// TIA Portal project "Lab1" (V15)

(* hardware
DEVICE "S7-1200 station_1"  S7-1200 Station
   slot 0: "Rack_0"  S7-1200 Rack  Rack  V1.0
   slot 1: "PLC_1"  CPU 1214C AC/DC/Rly  6ES7 214-1BG40-0XB0  V4.2
DEVICE "HMI_1"  KTP1000 Basic color PN
   slot 0: "HMI_1"  KTP1000 Basic color PN  6AV6 647-0AF11-3AX0  12.0.0.0
   slot 1: "HMI_RT_1"  KTP1000 Basic color PN  6AV6 647-0AF11-3AX0  12.0.0.0
   slot 5: "HMI_1.IE_CP_1"  PROFINET Interface  12.0.0.0
      slot 1: "PROFINET Interface_1"  PROFINET Interface
         slot 1: "Port_1"  Port
*)

// ===== PLC "PLC_1"  CPU 1214C AC/DC/Rly =====

VAR_GLOBAL   // PLC tag table "Default tag table"
   "Start_NC" AT %M4.0 : Bool;
   "Manual_NO" AT %I0.2 : Bool;
   "Auto_NO" AT %I0.3 : Bool;
   "Stop_NC" AT %M4.1 : Bool;
   "SigSklop_NC" AT %I0.6 : Bool;
   "Bimetal_NC" AT %I0.7 : Bool;
   "Prekostruj_NO" AT %I1.0 : Bool;
   "Kontaktor_NO" AT %I1.1 : Bool;
   "Zelena" AT %Q0.0 : Bool;
   "Crvena" AT %Q0.1 : Bool;
   "Kontaktor" AT %Q0.2 : Bool;
   "Clock_Byte" AT %MB53 : Byte;
   "Clock_10Hz" AT %M53.0 : Bool;
   "Clock_5Hz" AT %M53.1 : Bool;
   "Clock_2.5Hz" AT %M53.2 : Bool;
   "Clock_2Hz" AT %M53.3 : Bool;
   "Clock_1.25Hz" AT %M53.4 : Bool;
   "Clock_1Hz" AT %M53.5 : Bool;
   "Clock_0.625Hz" AT %M53.6 : Bool;
   "Clock_0.5Hz" AT %M53.7 : Bool;
   "Blink" AT %M3.2 : Bool;
   "Blink_FF" AT %M3.1 : Bool;
   "Blink_Pulse" AT %M3.0 : Bool;
   "Auto_Stanje_FF" AT %M2.0 : Bool;
   "Greska" AT %M0.4 : Bool;
   "Greska_Bimetal" AT %M0.0 : Bool;
   "Greska_Prekostruj" AT %M0.1 : Bool;
   "Greska_Kontaktor" AT %M0.2 : Bool;
   "Greska_Svestop" AT %M0.3 : Bool;
   "Cekamo" AT %M2.2 : Bool;
   "Blink_Cnt_Greska_Pos" AT %M3.3 : Bool;
   "Blink_FF_Greska_Pos" AT %M3.4 : Bool;
   "OFF_NO" AT %M2.1 : Bool;
   "Bimetal_FF" AT %M1.0 : Bool;
   "Prekostruj_FF" AT %M1.1 : Bool;
   "Svestop_FF" AT %M1.3 : Bool;
   "GKontaktor_FF" AT %M1.2 : Bool;
   "Cekamo_Trig_P" AT %M2.3 : Bool;
   "Cekamo_Trig_N" AT %M2.4 : Bool;
   "Ocekivani_Kontaktor" AT %M2.5 : Bool;
   "Start_Taster_NC" AT %I0.0 : Bool;
   "Stop_Taster_NC" AT %I0.4 : Bool;
   "Start_HMI_NO" AT %M4.2 : Bool;
   "Stop_HMI_NO" AT %M4.3 : Bool;
   "ManualYES" AT %M4.4 : Bool;
   "AlarmWord" AT %MW0 : Word;
END_VAR

// folder: System blocks/Program resources

DATA_BLOCK "Counter_Blink"   // DB1
{ S7_Optimized_Access := 'TRUE' }
AUTHOR : Simatic
FAMILY : IEC
NAME : CNTR
VERSION : 1.0
// stored: InstanceOfName IEC_COUNTER
"IEC_COUNTER"
BEGIN
END_DATA_BLOCK

DATA_BLOCK "Timer_Start"   // DB2
{ S7_Optimized_Access := 'TRUE' }
AUTHOR : Simatic
FAMILY : IEC
NAME : IEC_TMR
VERSION : 1.0
// stored: InstanceOfName IEC_TIMER
"IEC_TIMER"
BEGIN
END_DATA_BLOCK

DATA_BLOCK "Timer_Cekamo"   // DB3
{ S7_Optimized_Access := 'TRUE' }
AUTHOR : Simatic
FAMILY : IEC
NAME : IEC_TMR
VERSION : 1.0
// stored: InstanceOfName IEC_TIMER
"IEC_TIMER"
BEGIN
END_DATA_BLOCK

// folder: (top level)

ORGANIZATION_BLOCK "Main"   // OB1, LAD, ProgramCycle
TITLE = "Main Program Sweep (Cycle)"
{ S7_Optimized_Access := 'TRUE' }
VERSION : 0.1
   VAR_INPUT
      Initial_Call : Bool;   // Initial call of this OB
      Remanence : Bool;   // =True, if remanent data are available
   END_VAR
   VAR_TEMP   // added for the SCL form of the ladder/FBD networks
      _w1 : Bool;
      _w2 : Bool;
      _w3 : Bool;
      _w4 : Bool;
   END_VAR
BEGIN

REGION Network 1: HMI stvari
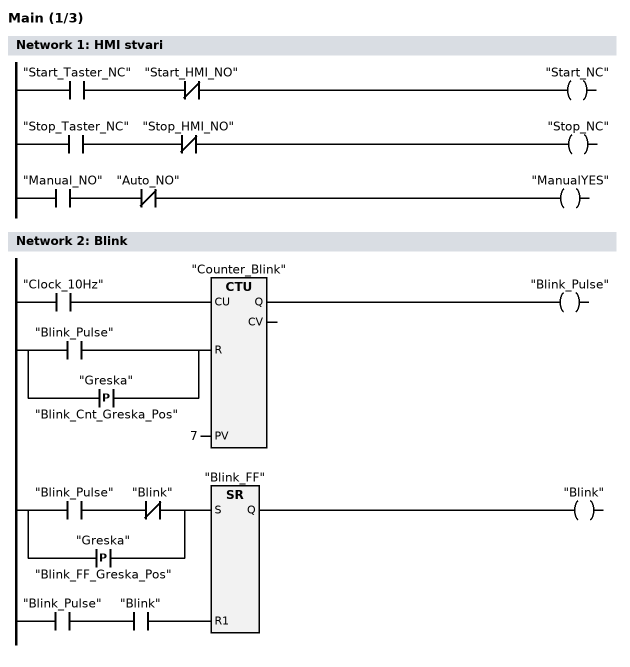
   RUNG wire#powerrail
      Contact( "Start_Taster_NC" )
      I_Contact( "Start_HMI_NO" )
      Coil( "Start_NC" )
   END_RUNG
   RUNG wire#powerrail
      Contact( "Stop_Taster_NC" )
      I_Contact( "Stop_HMI_NO" )
      Coil( "Stop_NC" )
   END_RUNG
   RUNG wire#powerrail
      Contact( "Manual_NO" )
      I_Contact( "Auto_NO" )
      Coil( "ManualYES" )
   END_RUNG
   // the same network as SCL:
   "Start_NC" := "Start_Taster_NC" AND NOT "Start_HMI_NO";
   "Stop_NC" := "Stop_Taster_NC" AND NOT "Stop_HMI_NO";
   "ManualYES" := "Manual_NO" AND NOT "Auto_NO";
END_REGION

REGION Network 2: Blink
   #_w1 := "Greska" AND NOT "Blink_Cnt_Greska_Pos";   // rising edge of "Greska"
   "Blink_Cnt_Greska_Pos" := "Greska";
   "Counter_Blink".CTU(CU := "Clock_10Hz", R := "Blink_Pulse" OR #_w1, PV := 7);
   "Blink_Pulse" := "Counter_Blink".Q;
   #_w2 := "Greska" AND NOT "Blink_FF_Greska_Pos";   // rising edge of "Greska"
   "Blink_FF_Greska_Pos" := "Greska";
   IF ("Blink_Pulse" AND NOT "Blink") OR #_w2 THEN
       "Blink_FF" := TRUE;   // SR flip-flop
   END_IF;
   IF "Blink_Pulse" AND "Blink" THEN "Blink_FF" := FALSE; END_IF;
   "Blink" := "Blink_FF";
END_REGION

REGION Network 3: Detekcija greske na kontaktoru
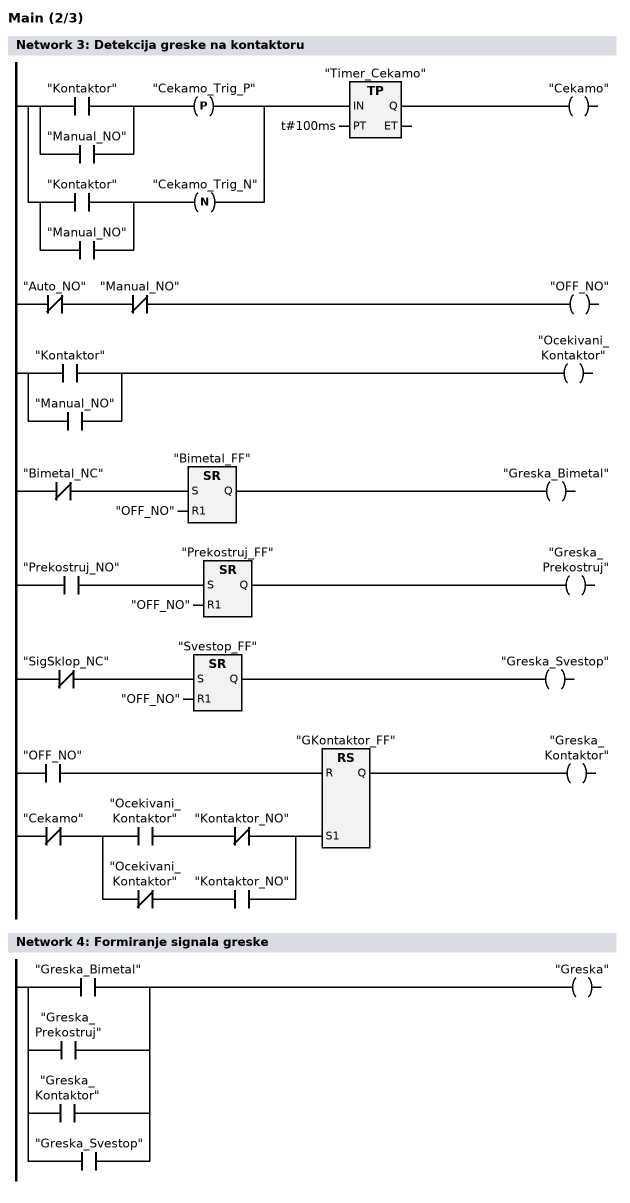
   #_w1 := "Kontaktor" OR "Manual_NO";
   #_w2 := #_w1 AND NOT "Cekamo_Trig_P";   // rising edge
   "Cekamo_Trig_P" := #_w1;
   #_w3 := "Kontaktor" OR "Manual_NO";
   #_w4 := NOT #_w3 AND "Cekamo_Trig_N";   // falling edge
   "Cekamo_Trig_N" := #_w3;
   "Timer_Cekamo".TP(IN := #_w2 OR #_w4, PT := t#100ms);
   "Cekamo" := "Timer_Cekamo".Q;
   "OFF_NO" := NOT "Auto_NO" AND NOT "Manual_NO";
   "Ocekivani_Kontaktor" := "Kontaktor" OR "Manual_NO";
   IF NOT "Bimetal_NC" THEN
       "Bimetal_FF" := TRUE;   // SR flip-flop
   END_IF;
   IF "OFF_NO" THEN "Bimetal_FF" := FALSE; END_IF;
   "Greska_Bimetal" := "Bimetal_FF";
   IF "Prekostruj_NO" THEN
       "Prekostruj_FF" := TRUE;   // SR flip-flop
   END_IF;
   IF "OFF_NO" THEN "Prekostruj_FF" := FALSE; END_IF;
   "Greska_Prekostruj" := "Prekostruj_FF";
   IF NOT "SigSklop_NC" THEN
       "Svestop_FF" := TRUE;   // SR flip-flop
   END_IF;
   IF "OFF_NO" THEN "Svestop_FF" := FALSE; END_IF;
   "Greska_Svestop" := "Svestop_FF";
   IF "OFF_NO" THEN
       "GKontaktor_FF" := FALSE;   // RS flip-flop
   END_IF;
   IF NOT "Cekamo" AND (("Ocekivani_Kontaktor" AND NOT "Kontaktor_NO") OR (NOT "Ocekivani_Kontaktor" AND "Kontaktor_NO")) THEN
       "GKontaktor_FF" := TRUE;
   END_IF;
   "Greska_Kontaktor" := "GKontaktor_FF";
END_REGION

REGION Network 4: Formiranje signala greske
   RUNG wire#powerrail
      Contact( "Greska_Bimetal" )
      wire#w1
      Coil( "Greska" )
   END_RUNG
   RUNG wire#powerrail
      Contact( "Greska_Prekostruj" )
   END_RUNG wire#w1
   RUNG wire#powerrail
      Contact( "Greska_Kontaktor" )
   END_RUNG wire#w1
   RUNG wire#powerrail
      Contact( "Greska_Svestop" )
   END_RUNG wire#w1
   // the same network as SCL:
   "Greska" := "Greska_Bimetal" OR "Greska_Prekostruj" OR "Greska_Kontaktor" OR "Greska_Svestop";
END_REGION

REGION Network 5: Auto dugmad
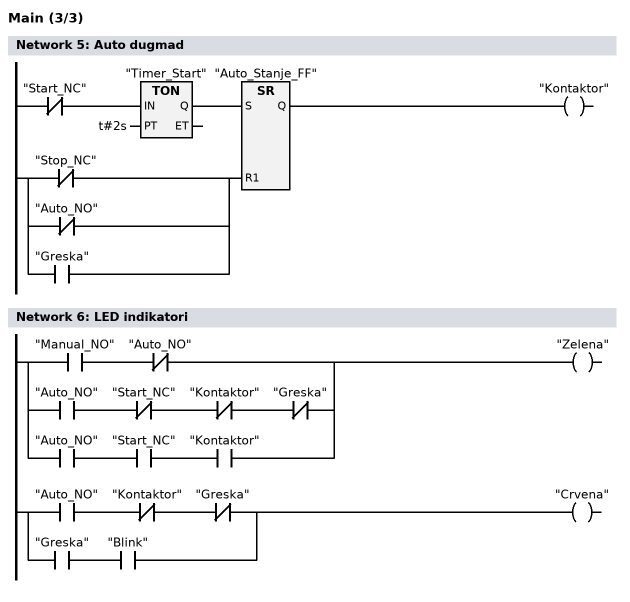
   "Timer_Start".TON(IN := NOT "Start_NC", PT := t#2s);
   IF "Timer_Start".Q THEN
       "Auto_Stanje_FF" := TRUE;   // SR flip-flop
   END_IF;
   IF NOT "Stop_NC" OR NOT "Auto_NO" OR "Greska" THEN "Auto_Stanje_FF" := FALSE; END_IF;
   "Kontaktor" := "Auto_Stanje_FF";
END_REGION

REGION Network 6: LED indikatori
   RUNG wire#powerrail
      Contact( "Manual_NO" )
      I_Contact( "Auto_NO" )
      wire#w1
      Coil( "Zelena" )
   END_RUNG
   RUNG wire#powerrail
      Contact( "Auto_NO" )
      I_Contact( "Start_NC" )
      I_Contact( "Kontaktor" )
      I_Contact( "Greska" )
   END_RUNG wire#w1
   RUNG wire#powerrail
      Contact( "Auto_NO" )
      Contact( "Start_NC" )
      Contact( "Kontaktor" )
   END_RUNG wire#w1
   RUNG wire#powerrail
      Contact( "Auto_NO" )
      I_Contact( "Kontaktor" )
      I_Contact( "Greska" )
      wire#w2
      Coil( "Crvena" )
   END_RUNG
   RUNG wire#powerrail
      Contact( "Greska" )
      Contact( "Blink" )
   END_RUNG wire#w2
   // the same network as SCL:
   "Zelena" := ("Manual_NO" AND NOT "Auto_NO") OR ("Auto_NO" AND NOT "Start_NC" AND NOT "Kontaktor" AND NOT "Greska") OR ("Auto_NO" AND "Start_NC" AND "Kontaktor");
   "Crvena" := ("Auto_NO" AND NOT "Kontaktor" AND NOT "Greska") OR ("Greska" AND "Blink");
END_REGION
END_ORGANIZATION_BLOCK

(* ===== HMI "HMI_RT_1" =====
system functions are stored by id; their names below are inferred from use
connection "HMI_Connection_1": ETHERNET, SMART_S7_1200_OMS

HMI tags "Default tag table"
   "Start_HMI_NO" : Bool = PLC Start_HMI_NO AT %M4.2, 100 ms
   "Stop_HMI_NO" : Bool = PLC Stop_HMI_NO AT %M4.3, 100 ms
   "Auto_NO" : Bool = PLC Auto_NO AT %I0.3, 100 ms
   "OFF_NO" : Bool = PLC OFF_NO AT %M2.1, 100 ms
   "Crvena" : Bool = PLC Crvena AT %Q0.1, 100 ms
   "Zelena" : Bool = PLC Zelena AT %Q0.0, 100 ms
   "ManualYES" : Bool = PLC ManualYES AT %M4.4, 100 ms
   "AlarmWord" : Word = PLC AlarmWord AT %MW0, 100 ms

discrete alarms
   1: 'Prekostrujna zaštita aktivirana.', class Warnings, trigger "AlarmWord" bit 1
   2: 'Bimetalna zaštita aktivirana.', class Warnings, trigger "AlarmWord" bit 0
   3: 'Desila se greška na kontaktoru.', class Warnings, trigger "AlarmWord" bit 2
   4: 'Svestop dugme pritisnuto.', class Warnings, trigger "AlarmWord" bit 3

Template "Template_1" 640x480
   Button "Exit" at 560,422 size 79x57; TextOff 'Exit'; PictureOff "ExitRuntime_KTP1000_Basic_color_PN"; PictureOn "ExitRuntime_KTP1000_Basic_color_PN"
      on Release: StopRuntime(0)
   Button "Template_Button" at 480,422 size 79x57; TextOff 'Text'
   Button "Template_Button_1" at 400,422 size 79x57; TextOff 'Text'
   Button "Template_Button_2" at 320,422 size 79x57; TextOff 'Text'
   Button "Template_Button_3" at 240,422 size 79x57; TextOff 'Text'
   Button "Template_Button_4" at 160,422 size 79x57; TextOff 'Text'
   Button "Template_Button_5" at 80,422 size 79x57; TextOff 'Text'
   Button "Alarms" at 0,422 size 79x57; TextOff 'Alarms'; PictureOff "AlarmDisplay_KTP1000_Basic_color_PN"; PictureOn "AlarmDisplay_KTP1000_Basic_color_PN"
      on Release: function_ef3f5d25("Alarm window_Unacknowledged", -1)

screen "Lol" 640x480, template "Template_1"
   Circle "Circle_1" at 50,50 size 100x100
      Appearance <- "Zelena"
   Circle "Circle_2" at 492,50 size 100x100
      Appearance <- "Crvena"
   TextField "Text field_1" at 400,281 size 31x18; Text 'MAN'
      Visibility <- "ManualYES"
   TextField "Text field_2" at 396,299 size 36x18; Text 'AUTO'
      Visibility <- "Auto_NO"
   TextField "Text field_3" at 404,317 size 23x18; Text 'OFF'
      Visibility <- "OFF_NO"
   TextField "Text field_4" at 203,299 size 43x18; Text 'MODE:'
   AlarmView "Alarm view_1" at 0,349 size 640x73
   Button "Button_1" at 150,232 size 96x32; TextOff 'Start'
      on Press: SetBit("Start_HMI_NO")
      on Release: ResetBit("Start_HMI_NO")
      Visibility <- "Auto_NO"
   Button "Button_2" at 396,232 size 96x32; TextOff 'Stop'
      on Press: SetBit("Stop_HMI_NO")
      on Release: ResetBit("Stop_HMI_NO")
      Visibility <- "Auto_NO"
*)